# EPICS autosave request: iocBoot/iocas/auto_settings.req
file "sample_settings.req", P=as:, N=sample_positioner
$(P)sample_positioner.PREC
